// TIA Portal V16 export
// export: Created 2021-11-12T13:32:34.5265801Z, ExportSetting WithDefaults, DisplayName Totally Integrated Automation Portal, DisplayVersion V16 Update 3, DisplayName TIA Portal Version Control Interface, DisplayVersion V16 Update 2, DisplayName TIA Portal Openness, DisplayVersion V16 Update 3, DisplayName SINAMICS Startdrive Advanced, DisplayVersion V16 Update 5, DisplayName SINAMICS Startdrive G130, G150, S120, S150, SINAMICS MV, S210, DisplayVersion V16 Update 5, DisplayName SINAMICS Startdrive G110M, G120, G120C, G120D, G120P, G115D, DisplayVersion V16 Update 5, DisplayName STEP 7 Professional, DisplayVersion V16 Update 3, DisplayName STEP 7 Safety, DisplayVersion V16, DisplayName WinCC UA Professional, DisplayVersion V16 Update 3
DATA_BLOCK "HMI_PARAM_220"   // DB2105
{ S7_Optimized_Access := 'TRUE' }
VERSION : 0.1
// stored: AutoNumber false, DBAccessibleFromOPCUA true, IsOnlyStoredInLoadMemory false, IsRetainMemResEnabled false, IsWriteProtectedInAS false, MemoryReserve 100
   VAR
      xxxxx___BinarySensors___xxxxx : Byte;
      xxxxx___BinaryOthers___xxxxx : Byte;
      "UF01-SF02_14" : "UDT_CH_DI_Parameter";   // Dopravník Remote
      "UF01-SF02_24" : "UDT_CH_DI_Parameter";   // Dopravník Automat
      "UF01-SF03_14" : "UDT_CH_DI_Parameter";   // Dopravník Manuál Vzad
      "UF01-SF03_24" : "UDT_CH_DI_Parameter";   // Dopravník Manuál Vpřed
      "UF01-SF04_14" : "UDT_CH_DI_Parameter";   // Dopravník Start automat
      "UF01-SF05_12" : "UDT_CH_DI_Parameter";   // Dopravník Stop
      "UF01-SF07_14" : "UDT_CH_DI_Parameter";   // Bedna Žádost o výměnu
      "UF01-SF08_14" : "UDT_CH_DI_Parameter";   // Bedna Vyměněna
      "UC12-FC01_14" : "UDT_CH_DI_Parameter";   // 400V Dopravník ++220 ( L2) OK
      xxxxx___AnalogueSensors___xxxxx : Byte;
      xxxxx___Drives___xxxxx : Byte;
      GL01_MA01 : "UDT_Drive1_Parameter";   // Dopravník na ostřižky (L2) - motor
      UC12_TA01 : "UDT_SINAMICS_G120_Parameter";   // Dopravník na ostřižky (L2) - měnič G120
      xxxxx___Others___xxxxx : Byte;
      CL01 : "UDT_PartCounter_Parameter";   // Bedna na přířezy
      xxxxx___SensorAlarms___xxxxx : Byte;
      xxxxx___ProcessAlarms___xxxxx : Byte;
      CL01_Alarm : "UDT_DI_Mon_Parameter";   // CL01 - box full
   END_VAR
   VAR RETAIN
      CL01_Warn : "UDT_DI_Mon_Parameter";   // CL01 - box full
   END_VAR
   VAR
      xxxxx__SafetyAlarms__xxxxx { S7_SetPoint := 'True'} : Byte;
      ES : "UDT_DI_Mon_Parameter";   // E-stop
   END_VAR
BEGIN
   UC12_TA01.RefSpdP2000 := 1500.0;
   UC12_TA01.RefCurrP2002 := 2.6;
   UC12_TA01.RefTrqP2003 := 9.88;
   CL01_Warn.Func := 16#2;
END_DATA_BLOCK
